// SIMATIC STEP 7 (V5.x) project Desbobinador V0

SYMBOL_TABLE
"CONTADOR"	C 1	COUNTER	// Cuenta el numero de planchas cortadas
"DBSARTEN"	DB 1	DB 1	// Datos asociados a la desbobinación de sartenes
"DBCACEROLA"	DB 2	DB 2
"DBWOK"	DB 3	DB 3
"DBPAELLERA"	DB 4	DB 4
"DESBOBINADO"	FB 1	FB 1	// Función que se encarga del desbobinado
"CIZALLADO"	FB 2	FB 2	// Funcion que se encaga del cizallado de planchas
"CORTAR"	FC 1	FC 1	// Funcion de cortar las planchas
"PESAJE"	FC 2	FC 2	// Función de pesaje
"MODOS"	FC 3	FC 3	// Gestión de modos
"SCALE"	FC 105	FC 105	// Scaling Values
"PRESENCIA"	I 124.0	BOOL	// Sensor que indica si la bobina está siendo correctamente desbobinada
"SENSOR SARTEN"	I 124.1	BOOL	// Sensor que indica que la plancha ha llegado a la longitud de corte adecuada
"SENSOR CACEROLA"	I 124.2	BOOL	// Sensor que indica que la plancha ha llegado a la longitud de corte adecuada
"SENSOR WOK"	I 124.3	BOOL	// Sensor que indica que la plancha ha llegado a la longitud de corte adecuada
"SENSOR PAELLERA"	I 124.4	BOOL	// Sensor que indica que la plancha ha llegado a la longitud de corte adecuada
"BOBINA COLOCADA"	I 124.5	BOOL	// Sensor que detecta si una bobina ha sido puesta en su lugar para empezar proceso
"SENSOR ABAJO"	I 124.6	BOOL	// Sensor que detecta que la cuchilla de cizallado está abajo
"SENSOR ARRIBA"	I 124.7	BOOL	// Sensor que detecta que la cuchilla de cizallado está arriba
"EXPULSADA"	I 125.0	BOOL	// Sensor que detecta que la plancha recien cortada es expulsada
"MODO A"	I 125.1	BOOL	// Funcionamiento en modo A
"MODO B"	I 125.2	BOOL	// Funcionamiento en modo B
"PALET"	I 125.3	BOOL
"PON"	I 125.4	BOOL
"POFF"	I 125.5	BOOL
"SARTEN"	M 100.1	BOOL	// Peso que corresponde a la bobina para hacer sartenes
"CACEROLA"	M 100.2	BOOL	// Peso que corresponde a la bobina para hacer cacerolas
"WOK"	M 100.3	BOOL	// Peso que corresponde a la bobina para hacer woks
"PAELLERA"	M 100.4	BOOL	// Peso que corresponde a la bobina para hacer paelleras
"CORTADO"	M 100.5	BOOL	// Indica que una plancha ha sido cortada
"X0"	M 101.0	BOOL
"X1"	M 101.1	BOOL
"X2"	M 101.2	BOOL
"X3"	M 101.3	BOOL
"X4"	M 101.4	BOOL
"X5"	M 101.5	BOOL
"X6"	M 101.6	BOOL
"X7"	M 101.7	BOOL
"X8"	M 102.0	BOOL
"X10"	M 102.2	BOOL
"X11"	M 102.3	BOOL
"X20"	M 103.4	BOOL
"X21"	M 103.5	BOOL
"X22"	M 103.6	BOOL
"X23"	M 103.7	BOOL
"X24"	M 104.0	BOOL
"X25"	M 104.1	BOOL
"X30"	M 104.2	BOOL
"X60"	M 104.3	BOOL
"X61"	M 104.4	BOOL
"X62"	M 104.5	BOOL
""	M 104.6	BOOL
""	M 104.7	BOOL
""	M 105.0	BOOL
""	M 105.1	BOOL
""	M 105.2	BOOL
"X40"	M 105.7	BOOL
"X41"	M 106.0	BOOL
"X42"	M 106.1	BOOL
"X43"	M 106.2	BOOL
"X44"	M 106.3	BOOL
"X50"	M 106.7	BOOL
"X51"	M 107.0	BOOL
"X52"	M 107.1	BOOL
"X100"	M 107.2	BOOL
"X101"	M 107.3	BOOL
"X110"	M 107.4	BOOL
"X111"	M 107.5	BOOL
"X53"	M 107.6	BOOL
"X120"	M 107.7	BOOL
"ENDCOUNT"	M 108.0	BOOL	// Marca que avisa del final de la cuenta
"X123"	M 108.2	BOOL
"X124"	M 108.3	BOOL
"X122"	M 108.4	BOOL
"X121"	M 108.5	BOOL
"X54"	M 108.6	BOOL
"STBYDESBOB"	M 108.7	BOOL	// Indica el estado stby del FB1 (desbobinado)
"INIDESBOB"	M 109.0	BOOL	// FP para iniciar el FB1
"INICIZA"	M 109.1	BOOL	// FP para iniciar el FB2
"PLANCHAS"	MW 3	INT	// Numero de planchas por bobina
"OB1"	OB 1	OB 1	// Main programa
"OB100"	OB 100	OB 100	// Inicio del programa
"PESO"	PIW 751	INT	// Sensor de peso que pesa las bobinas
"CENTRO"	PIW 752	INT	// Medida actual del centro
"ABRIR MCENTRO"	Q 124.1	BOOL	// Salida que hace más grande el centro de sujeción de la bobina
"CERRAR MCENTRO"	Q 124.2	BOOL	// Salida que hace más pequeño el centro de sujeción de la bobina
"DESBOBINAR"	Q 124.3	BOOL	// Actuador que activa la rotación del centro
"EXPULSAR BOBINA"	Q 124.4	BOOL	// Actuador que expulsa el centro de la bobina una vez ha acabado de desbobinar
"BAJAR CUCHILLA"	Q 124.5	BOOL	// Baja la cuchilla, si está a 0 la cuchilla sube
"EXPULSAR PALET"	Q 124.6	BOOL	// Activa un piston que expulsa la plancgha de la zona de corte
"PRENSA"	Q 124.7	BOOL	// Activa la prensa
END_SYMBOL_TABLE

FUNCTION_BLOCK "DESBOBINADO"	// FB 1
TITLE = DESBOBINADO
VERSION : 0.1
VAR_INPUT
  SENSOR : BOOL ;
  PRESENCIA : BOOL ;
  CENTRO : INT ;
  bit_de_trabajo : BOOL ;
  MCENTRO : INT ;
  Contador : COUNTER ;
END_VAR
VAR_OUTPUT
  ABRIRMCENTRO : BOOL ;
  DESBOBINAR : BOOL ;
  bit_ok : BOOL ;
  bit_error : BOOL ;
END_VAR
VAR
  x31 : BOOL ;
  x32 : BOOL ;
  x33 : BOOL ;
  x34 : BOOL ;
  s1 : BOOL ;
END_VAR
VAR_TEMP
  watchdog_master : BOOL ;
END_VAR
BEGIN
NETWORK
TITLE = Arranque
      SET;
      FP    #bit_de_trabajo;
      S     #x31;
      R     #x32;
      R     #x33;
      R     #x34;
      R     #s1;
      R     #bit_error;
      R     #bit_ok;
NETWORK
TITLE = x31 a x32
//Comparacion medida centro con medida nominal del centro para pasar de x31 a x32
      A     #x31;
      A(;
      L     #CENTRO;
      L     #MCENTRO;
      ==R;
      );
      R     #x31;
      S     #x32;
NETWORK
TITLE = x32 a x33
//Presencia detecta que la plancha esta en posicion para empezar el proceso de 
//desbobinado-cizallado
      A     #x32;
      FP    #PRESENCIA;
      R     #x32;
      S     #x33;
NETWORK
TITLE = x33 a x34
//Detecta que la plancha esta lista para ser cizallada
      A     #x33;
      A     #SENSOR;
      R     #x33;
      S     #x34;
NETWORK
TITLE = x34 a x33
//si el contador no ha acabado
      A     #x34;
      T     LD 1;
      TAK;
      T     LD 5;
      L     #Contador;
      T     LW 9;
      L     LD 5;
      L     LD 1;
      A     C [LW 9];
      AN    #SENSOR;
      R     M 105.1;
      S     M 105.0;
NETWORK
TITLE = x34 a s1
//si el contador ha cabado
      A     #x34;
      T     LD 1;
      TAK;
      T     LD 5;
      L     #Contador;
      T     LW 9;
      L     LD 5;
      L     LD 1;
      AN    C [LW 9];
      AN    #SENSOR;
      R     #x34;
      S     #s1;
NETWORK
TITLE = Tratamiento de bit de fin
      A     #s1;
      =     #bit_ok;
NETWORK
TITLE = Abrir centro
      A     #x31;
      =     #ABRIRMCENTRO;
NETWORK
TITLE = Desbobinar
      A     M 104.7;
      =     #DESBOBINAR;
NETWORK
TITLE = Carga del contador en x32
//Aun no sabemos como cargar un valor distinto en función del modo de 
//funcionamiento
      A     #x32;
      L     C#100;
      T     LD 1;
      TAK;
      T     LD 5;
      L     #Contador;
      T     LW 9;
      L     LD 5;
      L     LD 1;
      S     C [LW 9];
NETWORK
TITLE = Resta del contador y salida del x33
      A     #x33;
      =     #DESBOBINAR;
END_FUNCTION_BLOCK

FUNCTION_BLOCK "CIZALLADO"	// FB 2
TITLE = CIZALLADO
VERSION : 0.1
VAR_INPUT
  ini : BOOL ;
  SENSOR : BOOL ;
  PLANCHAS : INT ;
END_VAR
VAR
  INICORTAR : BOOL ;
  CORTADO : BOOL ;
END_VAR
BEGIN
NETWORK
TITLE =
      A     "X40";
      A     #ini;
      R     "X40";
      S     "X41";
NETWORK
TITLE =
      A     "X41";
      A     #SENSOR;
      R     "X41";
      S     "X42";
NETWORK
TITLE =
      A     "X42";
      A     "CORTADO";
      R     "X42";
      S     "X43";
NETWORK
TITLE =
      A     "X43";
      AN    "CONTADOR";
      R     "X43";
      S     "X41";
NETWORK
TITLE =
      A     "X43";
      A     "CONTADOR";
      R     "X43";
      S     "X40";
NETWORK
TITLE =
      CALL  "CORTAR" (
           ini                      := #INICORTAR,
           SENSORABAJO              := "SENSOR ABAJO",
           SENSORARRIBA             := "SENSOR ARRIBA",
           EXPULSADA                := "EXPULSADA",
           BAJARCUCHILLA            := "BAJAR CUCHILLA",
           EXPULSARPLANCHA          := "EXPULSAR PALET",
           CORTADO                  := #CORTADO);
NETWORK
TITLE =
      A     "X42";
      A     "CORTADO";
      R     "X42";
      S     "X43";
NETWORK
TITLE =
      A     "X43";
      A     "ENDCOUNT";
      R     "X43";
      S     "X40";
NETWORK
TITLE =
      A     "X43";
      AN    "ENDCOUNT";
      R     "X43";
      S     "X41";
NETWORK
TITLE =
      A     "X42";
      A     "X50";
      FP    #INICORTAR;
NETWORK
TITLE = Cuenta el numero de planchas cortadas
      A     "X43";
      CU    "CONTADOR";
NETWORK
TITLE =
      A     "X43";
      R     "X54";
      S     "X50";
      R     #CORTADO;
END_FUNCTION_BLOCK

FUNCTION "CORTAR" : VOID	// FC 1
VERSION : 0.1
VAR_INPUT
  ini : BOOL ;
  SENSORABAJO : BOOL ;
  SENSORARRIBA : BOOL ;
  EXPULSADA : BOOL ;
END_VAR
VAR_OUTPUT
  BAJARCUCHILLA : BOOL ;
  EXPULSARPLANCHA : BOOL ;
  CORTADO : BOOL ;
END_VAR
BEGIN
NETWORK
TITLE =
      A     "X50";
      A     #ini;
      R     "X50";
      S     "X51";
NETWORK
TITLE =
      A     "X51";
      A     #SENSORABAJO;
      R     "X51";
      S     "X52";
NETWORK
TITLE =
      A     "X52";
      A     #SENSORARRIBA;
      R     "X52";
      S     "X53";
NETWORK
TITLE =
      A     "X53";
      A     #EXPULSADA;
      R     "X53";
      S     "X54";
NETWORK
TITLE =
      A     "X50";
      S     #CORTADO;
      R     #EXPULSARPLANCHA;
NETWORK
TITLE =
      A     "X51";
      S     #BAJARCUCHILLA;
      R     #CORTADO;
NETWORK
TITLE =
      A     "X52";
      R     #BAJARCUCHILLA;
NETWORK
TITLE =
      A     "X53";
      S     #EXPULSARPLANCHA;
NETWORK
TITLE =
      A     "X54";
      S     #CORTADO;
END_FUNCTION

FUNCTION "PESAJE" : VOID	// FC 2
TITLE = PESAJE
VERSION : 0.1
VAR_INPUT
  in : INT ;
END_VAR
VAR_IN_OUT
  SARTEN : BOOL ;
  CACEROLA : BOOL ;
  WOK : BOOL ;
  PAELLERA : BOOL ;
END_VAR
VAR_TEMP
  retFC105 : WORD ;
  PESO : REAL ;
END_VAR
BEGIN
NETWORK
TITLE =
      A     "X120";
      JNB   _001;
      CALL  "SCALE" (
           $1                       := #in,
           $2                       := L#1112014848,
           $3                       := L#0,
           $4                       := FALSE,
           $5                       := #retFC105,
           $6                       := #PESO);
_001: NOP   0;
NETWORK
TITLE =
      L     #PESO;
      L     "DBSARTEN".PESO;
      ==R;
      =     #SARTEN;
NETWORK
TITLE =
      L     #PESO;
      L     "DBCACEROLA".PESO;
      ==R;
      =     #CACEROLA;
NETWORK
TITLE =
      L     #PESO;
      L     "DBWOK".PESO;
      ==R;
      =     #WOK;
NETWORK
TITLE =
      L     #PESO;
      L     "DBPAELLERA".PESO;
      ==R;
      =     #PAELLERA;
END_FUNCTION

FUNCTION "MODOS" : VOID	// FC 3
VERSION : 0.1
VAR_INPUT
  MODO1 : BOOL ;
  MODO2 : BOOL ;
END_VAR
VAR_OUTPUT
  CONTADOR : INT ;
  PSARTEN : INT ;
  PCACEROLA : INT ;
  PWOK : INT ;
  PPAELLERA : INT ;
END_VAR
VAR_IN_OUT
  X60 : BOOL ;
  X61 : BOOL ;
  X62 : BOOL ;
END_VAR
BEGIN
NETWORK
TITLE =
      A     #X60;
      A     #MODO1;
      R     #X60;
      S     #X61;
NETWORK
TITLE =
      A     #X60;
      AN    #MODO1;
      R     #X61;
      S     #X60;
NETWORK
TITLE =
      A     #X60;
      A     #MODO2;
      R     #X60;
      S     #X62;
NETWORK
TITLE =
      A     #X62;
      AN    #MODO2;
      R     #X62;
      S     #X62;
NETWORK
TITLE = Numero de planchas por bobina
      A     #X61;
      L     #CONTADOR;
      OPN   DB 100;
      L     #PSARTEN;
      OPN   DB 100;
      L     #PCACEROLA;
      OPN   DB 110;
      L     #PWOK;
      OPN   DB 120;
      L     #PPAELLERA;
      OPN   DB 130;
NETWORK
TITLE =
      A     #X62;
      L     #CONTADOR;
      OPN   DB 200;
      L     #PSARTEN;
      OPN   DB 200;
      L     #PCACEROLA;
      OPN   DB 220;
      L     #PWOK;
      OPN   DB 240;
      L     #PPAELLERA;
      OPN   DB 260;
END_FUNCTION

// FC 105: know-how protected block, not included

DATA_BLOCK "DBSARTEN"	// DB 1
VERSION : 0.1
  STRUCT
   CENTRO : INT  := 50;	//Tamaño del centro de la bobina
   PESO : INT  := 100;	//Peso de la bobina
   SENSOR : BOOL ;	//Sensor que detecta la posIcion para cortar
   PESOBOOL : BOOL ;	//Sensor que dice si se ha detectado el peso de este tipo de bobina
  END_STRUCT ;	
BEGIN
   PESO := 100;
END_DATA_BLOCK

DATA_BLOCK "DBCACEROLA"	// DB 2
VERSION : 0.1
  STRUCT
   CENTRO : INT  := 60;	//Variable provisional
   PESO : INT  := 110;
   SENSOR : BOOL ;
   PESOBOOL : BOOL ;
  END_STRUCT ;	
BEGIN
   PESO := 110;
END_DATA_BLOCK

DATA_BLOCK "DBWOK"	// DB 3
VERSION : 0.1
  STRUCT
   CENTRO : INT  := 60;	//Variable provisional
   PESO : INT  := 120;
   SENSOR : BOOL ;
   PESOBOOL : BOOL ;
  END_STRUCT ;	
BEGIN
   PESO := 120;
END_DATA_BLOCK

DATA_BLOCK "DBPAELLERA"	// DB 4
VERSION : 0.1
  STRUCT
   CENTRO : INT  := 50;	//Variable provisional
   PESO : INT  := 130;
   SENSOR : BOOL ;
   PESOBOOL : BOOL ;
  END_STRUCT ;	
BEGIN
   PESO := 130;
END_DATA_BLOCK

DATA_BLOCK DB 5
VERSION : 0.0
"DESBOBINADO"
BEGIN
END_DATA_BLOCK

DATA_BLOCK DB 6
VERSION : 0.0
"CIZALLADO"
BEGIN
END_DATA_BLOCK

ORGANIZATION_BLOCK "OB1"	// OB 1
TITLE = "Main Program Sweep (Cycle)"
VERSION : 0.1
VAR_TEMP
  OB1_EV_CLASS : BYTE ;	//Bits 0-3 = 1 (Coming event), Bits 4-7 = 1 (Event class 1)
  OB1_SCAN_1 : BYTE ;	//1 (Cold restart scan 1 of OB 1), 3 (Scan 2-n of OB 1)
  OB1_PRIORITY : BYTE ;	//Priority of OB Execution
  OB1_OB_NUMBR : BYTE ;	//1 (Organization block 1, OB1)
  OB1_RESERVED_1 : BYTE ;	//Reserved for system
  OB1_RESERVED_2 : BYTE ;	//Reserved for system
  OB1_PREV_CYCLE : INT ;	//Cycle time of previous OB1 scan (milliseconds)
  OB1_MIN_CYCLE : INT ;	//Minimum cycle time of OB1 (milliseconds)
  OB1_MAX_CYCLE : INT ;	//Maximum cycle time of OB1 (milliseconds)
  OB1_DATE_TIME : DATE_AND_TIME ;	//Date and time OB1 started
END_VAR
BEGIN
NETWORK
TITLE =
      A     "X100";
      A     "PON";
      AN    "POFF";
      R     "X100";
      S     "X101";
NETWORK
TITLE =
      A     "X101";
      A     "POFF";
      R     "X101";
      S     "X100";
NETWORK
TITLE =
      A     "X0";
      A     "X101";
      AN    "X60";
      R     "X0";
      S     "X1";
      S     "X10";
      S     "X20";
NETWORK
TITLE =
      A     "X1";
      A     "BOBINA COLOCADA";
      R     "X1";
      S     "X2";
NETWORK
TITLE =
      A     "X2";
      A     "DBSARTEN".PESOBOOL;
      R     "X2";
      S     "X3";
NETWORK
TITLE =
      A     "X2";
      A     "DBCACEROLA".PESOBOOL;
      R     "X2";
      S     "X4";
NETWORK
TITLE =
      A     "X2";
      A     "DBWOK".PESOBOOL;
      R     "X2";
      S     "X5";
NETWORK
TITLE =
      A     "X2";
      A     "DBPAELLERA".PESOBOOL;
      R     "X2";
      S     "X6";
NETWORK
TITLE =
      A     "X3";
      O     "X4";
      O     "X5";
      O     "X6";
      R     "X121";
      R     "X122";
      R     "X123";
      R     "X124";
      S     "X120";
NETWORK
TITLE =
      A(;
      A     "X3";
      O     "X4";
      O     "X5";
      O     "X6";
      );
      A     "X30";
      R     "X3";
      R     "X4";
      R     "X5";
      R     "X6";
      S     "X7";
NETWORK
TITLE =
      A     "X7";
      A(;
      L     PIW 753;
      L     0;
      ==R;
      );
      R     "X7";
      S     "X8";
NETWORK
TITLE =
      A     "X8";
      A     "X101";
      AN    "BOBINA COLOCADA";
      R     "X8";
      S     "X1";
NETWORK
TITLE =
      A     "X10";
      A     "DESBOBINAR";
      A     "X101";
      R     "X10";
      S     "X11";
NETWORK
TITLE =
      A     "X20";
      A     "DBSARTEN".PESOBOOL;
      R     "X20";
      S     "X21";
NETWORK
TITLE =
      A     "X20";
      A     "DBCACEROLA".PESOBOOL;
      R     "X20";
      S     "X22";
NETWORK
TITLE =
      A     "X20";
      A     "DBWOK".PESOBOOL;
      R     "X20";
      S     "X23";
NETWORK
TITLE =
      A     "X20";
      A     "DBPAELLERA".PESOBOOL;
      R     "X20";
      S     "X24";
      A     "X40";
NETWORK
TITLE =
      A(;
      A     "X21";
      O     "X22";
      O     "X23";
      O     "X24";
      );
      A     "X30";
      R     "X21";
      R     "X22";
      R     "X23";
      R     "X24";
      S     "X25";
NETWORK
TITLE =
      A     "X25";
      A     "X101";
      AN    "PALET";
      R     "X25";
      S     "X20";
NETWORK
TITLE =
      A(;
      A     "X8";
      AN    "BOBINA COLOCADA";
      );
      A     "X10";
      A(;
      A     "X25";
      AN    "PALET";
      );
      A     "X100";
      R     "X8";
      R     "X10";
      R     "X25";
      S     "X0";
NETWORK
TITLE =
      A     "X0";
      CALL  "MODOS" (
           MODO1                    := "MODO A",
           MODO2                    := "MODO B",
           CONTADOR                 := "PLANCHAS",
           PSARTEN                  := "DBSARTEN".PESO,
           PCACEROLA                := "DBCACEROLA".PESO,
           PWOK                     := "DBWOK".PESO,
           PPAELLERA                := "DBPAELLERA".PESO,
           X60                      := "X60",
           X61                      := "X61",
           X62                      := "X62");
NETWORK
TITLE =
      A     "X2";
      CALL  "PESAJE" (
           in                       := "CENTRO",
           SARTEN                   := "DBSARTEN".PESOBOOL,
           CACEROLA                 := "DBCACEROLA".PESOBOOL,
           WOK                      := "DBWOK".PESOBOOL,
           PAELLERA                 := "DBPAELLERA".PESOBOOL);
NETWORK
TITLE = Salida que hace más pequeño el centro de sujeción de la bobina
      A     "X7";
      S     "CERRAR MCENTRO";
NETWORK
TITLE = Salida que hace más pequeño el centro de sujeción de la bobina
      A     "X8";
      R     "CERRAR MCENTRO";
      S     "EXPULSAR BOBINA";
NETWORK
TITLE = Activa la prensa
      A     "X11";
      S     "PRENSA";
NETWORK
TITLE = Activa la prensa
      A     "X10";
      R     "PRENSA";
NETWORK
TITLE = Activa un piston que expulsa la plancgha de la zona de corte
      A     "X20";
      R     "EXPULSAR PALET";
NETWORK
TITLE = Activa un piston que expulsa la plancgha de la zona de corte
      A     "X25";
      S     "EXPULSAR PALET";
NETWORK
TITLE =
      A     "X2";
      BLD   3;
      =     L 24.0;
      CDB;
      OPN   DI 5;
      TAR2  LD 20;
      OPN   DI 1;
      A     DIX 4.0;
      OPN   DI 5;
      =     DIX 0.0;
      A     "PRESENCIA";
      =     DIX 0.1;
      OPN   DI 1;
      L     DIW 0;
      OPN   DI 5;
      T     DIW 2;
      L     "PLANCHAS";
      T     DIW 4;
      A     "INIDESBOB";
      =     DIX 6.0;
      L     "CENTRO";
      T     DIW 8;
      LAR2  P#DBX 0.0;
      UC    "DESBOBINADO";
      LAR2  LD 20;
      A     DIX 10.0;
      =     "ABRIR MCENTRO";
      A     DIX 10.1;
      =     "CERRAR MCENTRO";
      A     DIX 10.2;
      =     "DESBOBINAR";
      A     DIX 10.3;
      =     "STBYDESBOB";
      CDB;
      BLD   4;
      FP    "INIDESBOB";
NETWORK
TITLE =
      A     "X3";
      BLD   3;
      =     L 24.0;
      CDB;
      OPN   DI 5;
      TAR2  LD 20;
      OPN   DI 2;
      A     DIX 4.0;
      OPN   DI 5;
      =     DIX 0.0;
      A     "PRESENCIA";
      =     DIX 0.1;
      OPN   DI 2;
      L     DIW 0;
      OPN   DI 5;
      T     DIW 2;
      L     "PLANCHAS";
      T     DIW 4;
      A     "INIDESBOB";
      =     DIX 6.0;
      L     "CENTRO";
      T     DIW 8;
      LAR2  P#DBX 0.0;
      UC    "DESBOBINADO";
      LAR2  LD 20;
      A     DIX 10.0;
      =     "ABRIR MCENTRO";
      A     DIX 10.1;
      =     "CERRAR MCENTRO";
      A     DIX 10.2;
      =     "DESBOBINAR";
      A     DIX 10.3;
      =     "STBYDESBOB";
      CDB;
      BLD   4;
      FP    "INIDESBOB";
NETWORK
TITLE =
      A     "X5";
      BLD   3;
      =     L 24.0;
      CDB;
      OPN   DI 5;
      TAR2  LD 20;
      OPN   DI 3;
      A     DIX 4.0;
      OPN   DI 5;
      =     DIX 0.0;
      A     "PRESENCIA";
      =     DIX 0.1;
      OPN   DI 3;
      L     DIW 0;
      OPN   DI 5;
      T     DIW 2;
      L     "PLANCHAS";
      T     DIW 4;
      A     "INIDESBOB";
      =     DIX 6.0;
      L     "CENTRO";
      T     DIW 8;
      LAR2  P#DBX 0.0;
      UC    "DESBOBINADO";
      LAR2  LD 20;
      A     DIX 10.0;
      =     "ABRIR MCENTRO";
      A     DIX 10.1;
      =     "CERRAR MCENTRO";
      A     DIX 10.2;
      =     "DESBOBINAR";
      A     DIX 10.3;
      =     "STBYDESBOB";
      CDB;
      BLD   4;
      FP    "INIDESBOB";
NETWORK
TITLE =
      A     "X6";
      BLD   3;
      =     L 24.0;
      CDB;
      OPN   DI 5;
      TAR2  LD 20;
      OPN   DI 4;
      A     DIX 4.0;
      OPN   DI 5;
      =     DIX 0.0;
      A     "PRESENCIA";
      =     DIX 0.1;
      OPN   DI 4;
      L     DIW 0;
      OPN   DI 5;
      T     DIW 2;
      L     "PLANCHAS";
      T     DIW 4;
      A     "INIDESBOB";
      =     DIX 6.0;
      L     "CENTRO";
      T     DIW 8;
      LAR2  P#DBX 0.0;
      UC    "DESBOBINADO";
      LAR2  LD 20;
      A     DIX 10.0;
      =     "ABRIR MCENTRO";
      A     DIX 10.1;
      =     "CERRAR MCENTRO";
      A     DIX 10.2;
      =     "DESBOBINAR";
      A     DIX 10.3;
      =     "STBYDESBOB";
      CDB;
      BLD   4;
      FP    "INIDESBOB";
NETWORK
TITLE =
      A     "X21";
      CALL  "CIZALLADO" , DB 6 (
           ini                      := "INICIZA",
           SENSOR                   := "DBSARTEN".SENSOR,
           PLANCHAS                 := "PLANCHAS");
      FP    "INICIZA";
NETWORK
TITLE =
      A     "X22";
      CALL  "CIZALLADO" , DB 6 (
           ini                      := "INICIZA",
           SENSOR                   := "DBCACEROLA".SENSOR,
           PLANCHAS                 := "PLANCHAS");
      FP    "INICIZA";
NETWORK
TITLE =
      A     "X23";
      CALL  "CIZALLADO" , DB 6 (
           ini                      := "INICIZA",
           SENSOR                   := "DBCACEROLA".SENSOR,
           PLANCHAS                 := "PLANCHAS");
      FP    "INICIZA";
NETWORK
TITLE =
      A     "X23";
      CALL  "CIZALLADO" , DB 6 (
           ini                      := "INICIZA",
           SENSOR                   := "DBWOK".SENSOR,
           PLANCHAS                 := "PLANCHAS");
      FP    "INICIZA";
NETWORK
TITLE =
      A     "X24";
      CALL  "CIZALLADO" , DB 6 (
           ini                      := "INICIZA",
           SENSOR                   := "DBPAELLERA".SENSOR,
           PLANCHAS                 := "PLANCHAS");
      FP    "INICIZA";
END_ORGANIZATION_BLOCK

ORGANIZATION_BLOCK "OB100"	// OB 100
TITLE = "Complete Restart"
VERSION : 0.1
VAR_TEMP
  OB100_EV_CLASS : BYTE ;	//16#13, Event class 1, Entering event state, Event logged in diagnostic buffer
  OB100_STRTUP : BYTE ;	//16#81/82/83/84 Method of startup
  OB100_PRIORITY : BYTE ;	//Priority of OB Execution
  OB100_OB_NUMBR : BYTE ;	//100 (Organization block 100, OB100)
  OB100_RESERVED_1 : BYTE ;	//Reserved for system
  OB100_RESERVED_2 : BYTE ;	//Reserved for system
  OB100_STOP : WORD ;	//Event that caused CPU to stop (16#4xxx)
  OB100_STRT_INFO : DWORD ;	//Information on how system started
  OB100_DATE_TIME : DATE_AND_TIME ;	//Date and time OB100 started
END_VAR
BEGIN
NETWORK
TITLE =
      SET;
      S     "X0";
      R     "X1";
      R     "X2";
      R     "X3";
      R     "X4";
      R     "X5";
      R     "X6";
      R     "X7";
      R     "X8";
      R     "X10";
      R     "X11";
      R     "X20";
      R     "X21";
      R     "X22";
      R     "X23";
      R     "X24";
      R     "X25";
      S     "X30";
      S     "X60";
      R     "X61";
      R     "X62";
      R     M 104.6;
      R     M 104.7;
      R     M 105.0;
      R     M 105.1;
      R     M 105.2;
      S     "X40";
      R     "X41";
      R     "X42";
      R     "X43";
      R     "X44";
      S     "X50";
      R     "X51";
      R     "X52";
      S     "X100";
      R     "X101";
      S     "X110";
      R     "X111";
      R     "X53";
      S     "X120";
      R     "ENDCOUNT";
      R     "X123";
      R     "X124";
      R     "X122";
      R     "X121";
      R     "X54";
      R     "STBYDESBOB";
      R     "INIDESBOB";
      R     "INICIZA";
      R     "SARTEN";
      R     "CACEROLA";
      R     "WOK";
      R     "PAELLERA";
      R     "CORTADO";
END_ORGANIZATION_BLOCK
